TYPE ST_Coordinate :
STRUCT
	fX				: REAL;
	fY				: REAL;
END_STRUCT
END_TYPE

(* stored: Version 1.1.0.1, ProductVersion 3.1.4022.9
   DUT ST_Coordinate: Id {e0942c10-88a6-4b13-bccd-26225784f780} *)
